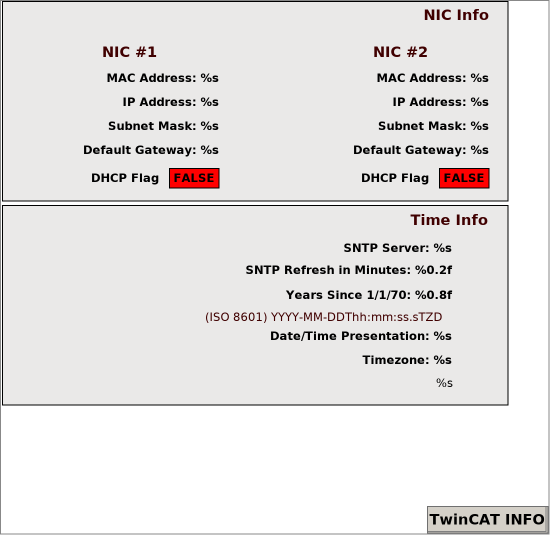
VISUALIZATION MDP_NicTime  // 550x535
    RoundedRectangle (2,1 506x200)
    Rectangle (7,67 215x22), "MAC Address: %s", text variable: System_Functions.ST_NIC0_ModContent.sMACAddress
    Rectangle (9,91 213x22), "IP Address: %s", text variable: System_Functions.ST_NIC0_ModContent.sIPAddress
    Rectangle (11,115 211x22), "Subnet Mask: %s", text variable: System_Functions.ST_NIC0_ModContent.sSubnetMask
    Rectangle (14,139 208x22), "Default Gateway: %s", text variable: System_Functions.ST_NIC0_ModContent.sDefaultGateway
    Group (169,168 50x20)
        Rectangle (0,0 50x20), "TRUE", invisible if: NOT System_Functions.ST_NIC0_ModContent.xDHCP
        Rectangle (0,0 50x20), "FALSE", invisible if: System_Functions.ST_NIC0_ModContent.xDHCP
    Label (77,166 85x24), "DHCP Flag"
    Rectangle (277,67 215x22), "MAC Address: %s", text variable: System_Functions.ST_NIC1_ModContent.sMACAddress
    Rectangle (279,91 213x22), "IP Address: %s", text variable: System_Functions.ST_NIC1_ModContent.sIPAddress
    Rectangle (281,115 211x22), "Subnet Mask: %s", text variable: System_Functions.ST_NIC1_ModContent.sSubnetMask
    Rectangle (284,139 208x22), "Default Gateway: %s", text variable: System_Functions.ST_NIC1_ModContent.sDefaultGateway
    Group (439,168 50x20)
        Rectangle (0,0 50x20), "TRUE", invisible if: NOT System_Functions.ST_NIC1_ModContent.xDHCP
        Rectangle (0,0 50x20), "FALSE", invisible if: System_Functions.ST_NIC1_ModContent.xDHCP
    Label (350,166 82x24), "DHCP Flag"
    Button (427,506 121x27), "TwinCAT INFO"
        OnMouseClick: change screen: TwinCAT_INFO
    Label (372,2 120x26), "NIC Info"
    Label (99,39 120x26), "NIC #1"
    Label (370,39 120x26), "NIC #2"
    RoundedRectangle (2,205 506x200)
    Label (371,207 120x26), "Time Info"
    Rectangle (10,237 445x22), "SNTP Server: %s", text variable: g_sHMI_SNTP_Server
    Rectangle (8,259 447x22), "SNTP Refresh in Minutes: %0.2f", text variable: g_lrHMI_SNTP_Refresh_Minutes
    Rectangle (10,284 445x22), "Years Since 1/1/70: %0.8f", text variable: g_lrHMI_Years_Since_1_1_1970
    Rectangle (9,325 446x22), "Date/Time Presentation: %s", text variable: System_Functions.ST_NIC0_ModContent.sMACAddress
    Rectangle (6,349 449x22), "Timezone: %s", text variable: System_Functions.ST_NIC0_ModContent.sMACAddress
    Label (202,304 274x26), "(ISO 8601) YYYY-MM-DDThh:mm:ss.sTZD"
    Rectangle (15,368 441x30), "%s", text variable: g_sHMI_CurrentTimeZone
END_VISUALIZATION

(* stored: Version 1.1.0.1, ProductVersion 3.1.0.18
   Visu MDP_NicTime: Id {1bd932f8-134d-436d-9579-59c84ea435c9} *)
